TYPE ST_VRC :
STRUCT
(* Readbacks *)
	//If True, Valve is Open
	i_xOpnLS	:	BOOL;
	//If True, Vavle is Closed
	i_xClsLS	:	BOOL;
	
	eState	:	E_ValvePositionState;

(* Inputs *)
	//Manually Pressing valve "Open/Close" on EDM
	xOPN_SW	: BOOL;
	//Manually toggling valve Local "ILK on button" on EDM
	xOvrdOpn	:	BOOL;
	//Calculated permissions to open valve
	xOPN_OK	: BOOL;
	//???
	xCLS_OK : BOOL := TRUE;
(* Outputs *)
	//When True, Opens valve
	//When False, Closes valve
	xOPN_DO	: BOOL;

END_STRUCT
END_TYPE

(* stored: Version 1.1.0.1, ProductVersion 3.1.4019.2
   DUT ST_VRC: Id {cb0eb88e-32ce-4b88-92df-8442dedadfcd} *)
